//{attribute 'qualified_only'}
//{attribute 'strict'}
TYPE E_EDM_Out :
(
	eEdmOut_none := 0,										(* Sicherheit | Rückmeldung | Xxx *)
	eEdmOut_Nothalt,

(*Maximum*)
	eEdmOut_nMaxIdx
);
END_TYPE

(* stored: Version 1.1.0.1, ProductVersion 3.1.4024.12
   DUT E_EDM_Out: Id {e6c94db3-0f0e-44d8-9c48-14f98c63444a} *)
